# EPICS StreamDevice protocol: protocols/dio432.proto
Terminator = LF;
ExtraInput = Ignore;

get_dpg {
	out "dpg_status";
	in "%d %(\$1)d";
}

getCosSta {
	out "status_latch";
	in "0x%(\$1:\$2)04x%(\$1:\$3)04x";
};

setCosEn {
	out "cos_en %(\$1:\$2)04x%(\$1:\$3)04x";
	in;
}

getInstDI {
	out "di_snoop  %(\$1:\$2)04x%(\$1:\$3)04x";
	in;
}
